// TIA Portal V17 export
// export: Created 2024-06-16T17:47:33.1888839Z, ExportSetting WithDefaults, DisplayName Totally Integrated Automation Portal, DisplayVersion V17, DisplayName TIA Portal Openness, DisplayVersion V17, DisplayName TIA Portal Version Control Interface, DisplayVersion V17, DisplayName STEP 7 Professional, DisplayVersion V17, DisplayName STEP 7 Safety, DisplayVersion V17, DisplayName WinCC Professional, DisplayVersion V17
FUNCTION_BLOCK "Obj_St4_FB"   // FB400, FBD
{ S7_Optimized_Access := 'TRUE' }
VERSION : 0.1
// stored: AutoNumber false, IsIECCheckEnabled false, IsRetainMemResEnabled false, MemoryReserve 100, SetENOAutomatically false, UDAEnableTagReadback false
   VAR
      Axe_X1 : Struct
         _ActPos : Real;
         _ActVel : Real;
         _Mode : Int;
         Home : Bool;
         Halt : Bool;
         Jog : Bool;
         MoveAbs : Bool;
         MoveRel : Bool;
         MoveVel : Bool;
         PowerOff : Bool;
         PowerOn : Bool;
         SensPos : Bool;
         SensNeg : Bool;
         xBusy : Bool;
         xHomed : Bool;
         xMoveAbsDone : Bool;
         xMoveRelDone : Bool;
         xPower : Bool;
      END_STRUCT;
      Axe_Y1 : Struct
         _ActPos : Real;
         _ActVel : Real;
         _Mode : Int;
         Home : Bool;
         Halt : Bool;
         Jog : Bool;
         MoveAbs : Bool;
         MoveRel : Bool;
         MoveVel : Bool;
         PowerOff : Bool;
         PowerOn : Bool;
         SensPos : Bool;
         SensNeg : Bool;
         xBusy : Bool;
         xHomed : Bool;
         xMoveAbsDone : Bool;
         xMoveRelDone : Bool;
         xPower : Bool;
      END_STRUCT;
      Axe_Y2 : Struct
         _ActPos : Real;
         _ActVel : Real;
         _Mode : Int;
         Home : Bool;
         Halt : Bool;
         Jog : Bool;
         MoveAbs : Bool;
         MoveRel : Bool;
         MoveVel : Bool;
         PowerOff : Bool;
         PowerOn : Bool;
         SensPos : Bool;
         SensNeg : Bool;
         xBusy : Bool;
         xHomed : Bool;
         xMoveAbsDone : Bool;
         xMoveRelDone : Bool;
         xPower : Bool;
      END_STRUCT;
      Prehenseur_Z2 : Struct
         _ActPos : Real;
         _ActVel : Real;
         _Mode : Int;
         Home : Bool;
         Halt : Bool;
         Jog : Bool;
         MoveAbs : Bool;
         MoveRel : Bool;
         MoveVel : Bool;
         PowerOff : Bool;
         PowerOn : Bool;
         SensPos : Bool;
         SensNeg : Bool;
         xBusy : Bool;
         xHomed : Bool;
         xMoveAbsDone : Bool;
         xMoveRelDone : Bool;
         xPower : Bool;
      END_STRUCT;
      Prehenseur_Z3 : Struct
         _ActPos : Real;
         _ActVel : Real;
         _Mode : Int;
         Home : Bool;
         Halt : Bool;
         Jog : Bool;
         MoveAbs : Bool;
         MoveRel : Bool;
         MoveVel : Bool;
         PowerOff : Bool;
         PowerOn : Bool;
         SensPos : Bool;
         SensNeg : Bool;
         xBusy : Bool;
         xHomed : Bool;
         xMoveAbsDone : Bool;
         xMoveRelDone : Bool;
         xPower : Bool;
      END_STRUCT;
   END_VAR
BEGIN

REGION Network 1: Station 4 (Marquage) - Axe X
   // //___ ModePose : 
   //          1 ---> Relative positioning
   //          2 ---> Absolute positioning
   //          3 ---> Not supported
   //          4 ---> Referencing - referencing point approach
   //          5 ---> Referencing - set referencing point
   //          6 ---> Traversing block (record mode)
   //          7 ---> Jog
   //          8 ---> Not supported
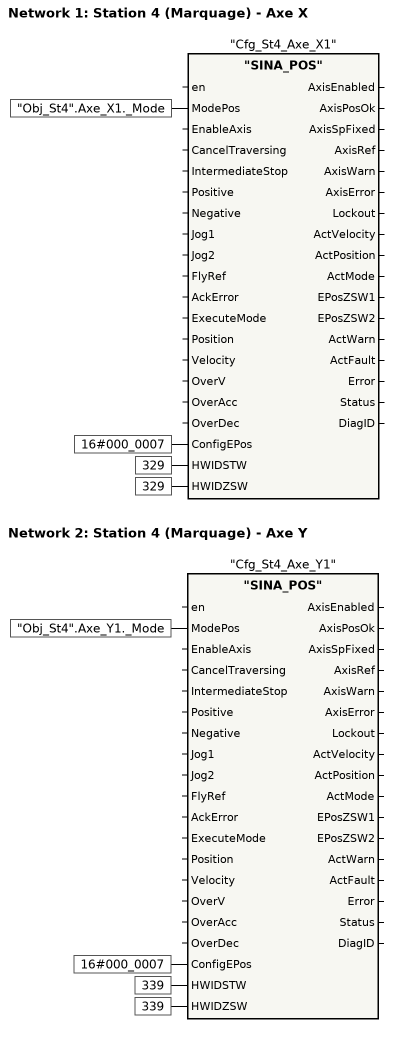
   "Cfg_St4_Axe_X1"(ModePos := "Obj_St4".Axe_X1._Mode,   // "SINA_POS"
                    ConfigEPos := 16#000_0007,
                    HWIDSTW := 329,
                    HWIDZSW := 329);
END_REGION

REGION Network 2: Station 4 (Marquage) - Axe Y
   // //___ ModePose : 
   //          1 ---> Relative positioning
   //          2 ---> Absolute positioning
   //          3 ---> Not supported
   //          4 ---> Referencing - referencing point approach
   //          5 ---> Referencing - set referencing point
   //          6 ---> Traversing block (record mode)
   //          7 ---> Jog
   //          8 ---> Not supported
   "Cfg_St4_Axe_Y1"(ModePos := "Obj_St4".Axe_Y1._Mode,   // "SINA_POS"
                    ConfigEPos := 16#000_0007,
                    HWIDSTW := 339,
                    HWIDZSW := 339);
END_REGION

REGION Network 3: Station 4 (Conforme) - Axe Y
   // //___ ModePose : 
   //          1 ---> Relative positioning
   //          2 ---> Absolute positioning
   //          3 ---> Not supported
   //          4 ---> Referencing - referencing point approach
   //          5 ---> Referencing - set referencing point
   //          6 ---> Traversing block (record mode)
   //          7 ---> Jog
   //          8 ---> Not supported
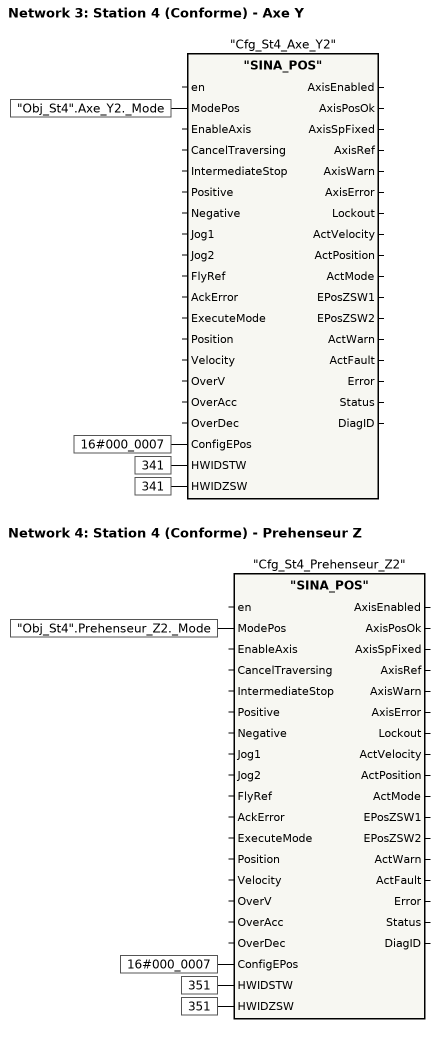
   "Cfg_St4_Axe_Y2"(ModePos := "Obj_St4".Axe_Y2._Mode,   // "SINA_POS"
                    ConfigEPos := 16#000_0007,
                    HWIDSTW := 341,
                    HWIDZSW := 341);
END_REGION

REGION Network 4: Station 4 (Conforme) - Prehenseur Z
   // //___ ModePose : 
   //          1 ---> Relative positioning
   //          2 ---> Absolute positioning
   //          3 ---> Not supported
   //          4 ---> Referencing - referencing point approach
   //          5 ---> Referencing - set referencing point
   //          6 ---> Traversing block (record mode)
   //          7 ---> Jog
   //          8 ---> Not supported
   "Cfg_St4_Prehenseur_Z2"(ModePos := "Obj_St4".Prehenseur_Z2._Mode,   // "SINA_POS"
                           ConfigEPos := 16#000_0007,
                           HWIDSTW := 351,
                           HWIDZSW := 351);
END_REGION

REGION Network 5: Station 4 (Non-Conforme) - Prehenseur Z
   // //___ ModePose : 
   //          1 ---> Relative positioning
   //          2 ---> Absolute positioning
   //          3 ---> Not supported
   //          4 ---> Referencing - referencing point approach
   //          5 ---> Referencing - set referencing point
   //          6 ---> Traversing block (record mode)
   //          7 ---> Jog
   //          8 ---> Not supported
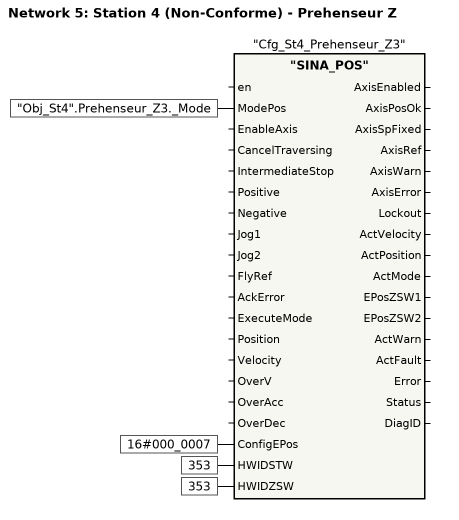
   "Cfg_St4_Prehenseur_Z3"(ModePos := "Obj_St4".Prehenseur_Z3._Mode,   // "SINA_POS"
                           ConfigEPos := 16#000_0007,
                           HWIDSTW := 353,
                           HWIDZSW := 353);
END_REGION
END_FUNCTION_BLOCK
